{attribute addProperty BoxType "EL2595-0000-0018"}
{attribute addProperty Id "ControlAT %Q*Control_659F2028162"}
{attribute addProperty CRC "1091680469"}
{attribute addProperty SizeInBites "16"}
{attribute addProperty SizeInBytes "2"}
TYPE DOX_Control_4111B8D5 :
STRUCT
	{attribute addProperty Name "Control"}
	Control AT %Q* : Control_659F2028;
END_STRUCT
END_TYPE

(* stored: Version 1.2.0.0, ProductVersion 3.1.4024.9
   DUT DOX_Control_4111B8D5: Id {8c0bdb4f-c69e-4c06-b384-b0c9aaecf515} *)
